FUNCTION_BLOCK FB_MotorJog EXTENDS FB_SolidSamplingModule
VAR_INPUT
END_VAR
VAR_OUTPUT
END_VAR
VAR
END_VAR

METHOD EnablePower : BOOL
VAR
	fbMC_Power	:	MC_Power;
END_VAR
// 
// process_gvl.fDecapperControl.Axis1.ReadStatus();
// 
// fbMC_Power(
// 	Axis:=process_gvl.fDecapperControl.Axis1, 
// 	Enable:=process_gvl.fDecapperControl.bEnable, 
// 	Status=> , 
// 	Busy=> , 
// 	Active=> , 
// 	Error=> , 
// 	ErrorID=> );
END_METHOD

METHOD MotorDosingPosition : BOOL
VAR_INPUT
END_VAR
END_METHOD

METHOD MotorLoadingPosition : BOOL
VAR_INPUT
END_VAR
END_METHOD

END_FUNCTION_BLOCK

(* stored: Version 1.1.0.1
   POU FB_MotorJog: Id {572e2650-5346-4e2a-bd24-17aaf2aabb29}, SpecialFunc None
   Method EnablePower: Id {bbd8026d-cdfa-44b8-9db6-db11045b5e31}
   Method MotorDosingPosition: Id {000e46a7-d768-4af3-a8d9-7f99c3aface3}
   Method MotorLoadingPosition: Id {e29b9f65-c08f-4666-b282-98670f3f7956} *)
